TYPE E_ValueDeviationStatus :
(
	OK,
	NOK
);
END_TYPE

(* stored: Version 1.1.0.1, ProductVersion 3.1.4024.13
   DUT E_ValueDeviationStatus: Id {e70155df-2dd5-03a4-0924-af611c1ce0ce} *)
